FUNCTION_BLOCK FB_Chiller
VAR_INPUT
END_VAR
VAR_OUTPUT
END_VAR
VAR
END_VAR

END_FUNCTION_BLOCK

(* stored: Version 1.1.0.1
   POU FB_Chiller: Id {ff4fd094-7be6-4b3f-8123-efaae2acfb8d}, SpecialFunc None *)
